FUNCTION_BLOCK SimpleMove_E
  (* Standard: 61499-2 *)
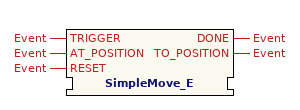
  EVENT_INPUT
    TRIGGER;
    AT_POSITION;
    RESET;
  END_EVENT
  EVENT_OUTPUT
    DONE;
    TO_POSITION;
  END_EVENT
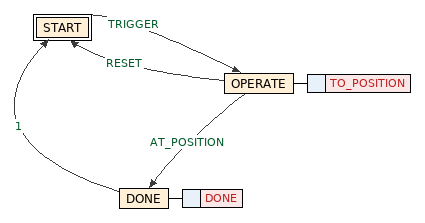
  EC_STATES
    START;
    OPERATE : -> TO_POSITION;
    DONE : -> DONE;
  END_STATES
  EC_TRANSITIONS
    START TO OPERATE := TRIGGER;
    OPERATE TO DONE := AT_POSITION;
    DONE TO START := 1;
    OPERATE TO START := RESET;
  END_TRANSITIONS
  ALGORITHM INIT IN ST:

  END_ALGORITHM
  ALGORITHM REQ IN ST:

  END_ALGORITHM
END_FUNCTION_BLOCK
